ABB RobotStudio station: RobotStudio.rsstnx

Station RobotStudio (saved by RobotStudio 23.3.10550.0)
Layout (positions relative to the parent item):
